Fanuc KAREL source: remote_gripper_info.kl

PROGRAM remotegripperinfo

%COMMENT = ' Remote Gripper Info'
%NOLOCKGROUP
%NOPAUSE=ERROR+COMMAND+TPENABLE
%NOBUSYLAMP

VAR
	response_file :FILE
	STATUS: INTEGER

	%INCLUDE ../core/core_gripper_info

BEGIN
	OPEN FILE response_file ('RW', 'RD:RESPONSE.HTM')
	STATUS = IO_STATUS(response_file)
	IF (STATUS <> 0) THEN
		RETURN
	ELSE
		CORE_GRIPPER_INFO(response_file)
	ENDIF

	CLOSE FILE response_file
END remotegripperinfo
